FUNCTION_BLOCK FB_RecipeBuilderWings EXTENDS FB_PackML_BaseModule IMPLEMENTS I_RecipeBuilder

VAR
    RecipeBuilder_HMI		: ST_RecipeBuilder_HMI;
    _Config                 : ST_RecipeBuilder_Config;
    _PanelFrontLength       : REAL;  
    _PanelFrontWidth        : REAL;      
    _PanelHeight            : REAL;    
    _RailHeightCorrection   : REAL;

    // --- NOWE ZMIENNE DO PRZECHOWYWANIA SEGMENTÓW ---
    _SegmentsCutX           : ARRAY [1..32] OF ST_CutSegment;
    _SegmentsCutY           : ARRAY [1..32] OF ST_CutSegment;
    _SegmentsGroove         : ARRAY [1..32] OF ST_CutSegment;
    _SegmentsToCutX         : INT;
    _SegmentsToCutY         : INT;
    _SegmentsToGroove       : INT;
END_VAR

METHOD Build : BOOL
VAR
    TotalY          : REAL;
    TotalX          : REAL;
    ShorterY        : REAL;
    ShorterX        : REAL;
    
    // Zmienna lokalna, dopóki nie dodasz jej do ST_RecipeBuilder_Config
    CuttingOverpass : REAL := 20.0; 
END_VAR

// Wyliczenia gabarytów na podstawie parametrów wejściowych (ze struktury _Config)
TotalY   := _Config.PanelFrontLength + 2 * _Config.PanelHeight;
TotalX   := _Config.PanelFrontWidht  + 2 * _Config.PanelHeight; // Uwaga na literówkę 'Widht' w strukturze!
ShorterY := TotalY - _Config.PanelHeight;
ShorterX := TotalX - _Config.PanelHeight;

// --- TRACE DLA WERYFIKACJI ---
Trace(Message:= CONCAT('--- BUILD BORGO WINGS START ---', ''));
Trace(Message:= CONCAT('Input PanelWidth: ', TO_STRING(_Config.PanelFrontWidht)));
Trace(Message:= CONCAT('Input PanelLength: ', TO_STRING(_Config.PanelFrontLength)));
Trace(Message:= CONCAT('Input PanelHeight: ', TO_STRING(_Config.PanelHeight)));
Trace(Message:= CONCAT('Calc TotalX: ', TO_STRING(TotalX)));
Trace(Message:= CONCAT('Calc TotalY: ', TO_STRING(TotalY)));
Trace(Message:= CONCAT('Calc ShorterX: ', TO_STRING(ShorterX)));
Trace(Message:= CONCAT('Calc ShorterY: ', TO_STRING(ShorterY)));

// ------------------------------------
// 1. Segregracja frezowania (Grooving)
// ------------------------------------
_SegmentsToGroove := 4;

_SegmentsGroove[1].Start.X := TotalX;
_SegmentsGroove[1].Stop.X  := 0;
_SegmentsGroove[1].Start.Y := ShorterY;
_SegmentsGroove[1].Stop.Y  := ShorterY;

_SegmentsGroove[2].Start.X := TotalX;
_SegmentsGroove[2].Stop.X  := 0; 
_SegmentsGroove[2].Start.Y := _Config.PanelHeight;
_SegmentsGroove[2].Stop.Y  := _Config.PanelHeight;

_SegmentsGroove[3].Start.X := ShorterX;
_SegmentsGroove[3].Stop.X  := ShorterX;
_SegmentsGroove[3].Start.Y := TotalY;
_SegmentsGroove[3].Stop.Y  := 0;

_SegmentsGroove[4].Start.Y := TotalY;
_SegmentsGroove[4].Stop.Y  := 0;
_SegmentsGroove[4].Start.X := _Config.PanelHeight;
_SegmentsGroove[4].Stop.X  := _Config.PanelHeight;

// ------------------------------------
// 2. Cięcie w osi X (Cut X)
// ------------------------------------
_SegmentsToCutX := 6;

// Short Box Segments
_SegmentsCutX[1].Start.X := TotalX + CuttingOverpass;
_SegmentsCutX[1].Stop.X  := ShorterX;
_SegmentsCutX[1].Start.Y := ShorterY;
_SegmentsCutX[1].Stop.Y  := ShorterY;

_SegmentsCutX[2].Start.X := _Config.PanelHeight;
_SegmentsCutX[2].Stop.X  := -CuttingOverpass;
_SegmentsCutX[2].Start.Y := ShorterY;
_SegmentsCutX[2].Stop.Y  := ShorterY;

_SegmentsCutX[3].Start.X := TotalX + CuttingOverpass;
_SegmentsCutX[3].Stop.X  := ShorterX;
_SegmentsCutX[3].Start.Y := _Config.PanelHeight;
_SegmentsCutX[3].Stop.Y  := _Config.PanelHeight;

_SegmentsCutX[4].Start.X := _Config.PanelHeight;
_SegmentsCutX[4].Stop.X  := -CuttingOverpass;
_SegmentsCutX[4].Start.Y := _Config.PanelHeight;
_SegmentsCutX[4].Stop.Y  := _Config.PanelHeight;

// Panel Dimensions Shorter Flaps
_SegmentsCutX[5].Start.X := TotalX + CuttingOverpass;
_SegmentsCutX[5].Stop.X  := -CuttingOverpass;
_SegmentsCutX[5].Start.Y := TotalY - _Config.RailHeightCorrection;
_SegmentsCutX[5].Stop.Y  := TotalY - _Config.RailHeightCorrection;

_SegmentsCutX[6].Start.X := TotalX + CuttingOverpass;
_SegmentsCutX[6].Stop.X  := -CuttingOverpass;
_SegmentsCutX[6].Start.Y := _Config.RailHeightCorrection;
_SegmentsCutX[6].Stop.Y  := _Config.RailHeightCorrection;

// ------------------------------------
// 3. Cięcie w osi Y (Cut Y)
// ------------------------------------
_SegmentsToCutY := 6;

// Short Box Segments
_SegmentsCutY[1].Start.X := ShorterX;
_SegmentsCutY[1].Stop.X  := ShorterX;
_SegmentsCutY[1].Start.Y := TotalY + CuttingOverpass;
_SegmentsCutY[1].Stop.Y  := ShorterY;

_SegmentsCutY[2].Start.X := _Config.PanelHeight;
_SegmentsCutY[2].Stop.X  := _Config.PanelHeight;
_SegmentsCutY[2].Start.Y := TotalY + CuttingOverpass;
_SegmentsCutY[2].Stop.Y  := ShorterY;

_SegmentsCutY[3].Start.X := ShorterX;
_SegmentsCutY[3].Stop.X  := ShorterX;
_SegmentsCutY[3].Start.Y := _Config.PanelHeight;
_SegmentsCutY[3].Stop.Y  := -CuttingOverpass;

_SegmentsCutY[4].Start.X := _Config.PanelHeight;
_SegmentsCutY[4].Stop.X  := _Config.PanelHeight;
_SegmentsCutY[4].Start.Y := _Config.PanelHeight;
_SegmentsCutY[4].Stop.Y  := -CuttingOverpass;

// Panel Dimensions
_SegmentsCutY[5].Start.X := TotalX;
_SegmentsCutY[5].Stop.X  := TotalX;
_SegmentsCutY[5].Start.Y := TotalY + CuttingOverpass;
_SegmentsCutY[5].Stop.Y  := -CuttingOverpass;

_SegmentsCutY[6].Start.X := 0;
_SegmentsCutY[6].Stop.X  := 0;
_SegmentsCutY[6].Start.Y := TotalY + CuttingOverpass;
_SegmentsCutY[6].Stop.Y  := -CuttingOverpass;

// Log podsumowujący ile odcinków wygenerowano
Trace(Message:= CONCAT('Segments Groove Count: ', TO_STRING(_SegmentsToGroove)));
Trace(Message:= CONCAT('Segments CutX Count: ', TO_STRING(_SegmentsToCutX)));
Trace(Message:= CONCAT('Segments CutY Count: ', TO_STRING(_SegmentsToCutY)));

//Zwracamy TRUE gdy budowanie się zakończyło
Build := TRUE;
END_METHOD

PROPERTY Config : ST_RecipeBuilder_Config
GET
Config := _Config;
END_GET
SET
RecipeBuilder_HMI.Config := Config;
END_SET
END_PROPERTY

// Provides interlocks for HMI control and updates HMI status information for this module
METHOD PROTECTED HMICommunication

// This method is called cyclically by CyclicLogic()
_PanelFrontWidth      := RecipeBuilder_HMI.Config.PanelFrontWidht;
_PanelFrontLength     := RecipeBuilder_HMI.Config.PanelFrontLength;
_PanelHeight          := RecipeBuilder_HMI.Config.PanelHeight;
_RailHeightCorrection := RecipeBuilder_HMI.Config.RailHeightCorrection;
END_METHOD

PROPERTY SegmentsCutX : REFERENCE TO ARRAY [1..32] OF ST_CutSegment
GET
SegmentsCutX REF= _SegmentsCutX;
END_GET
END_PROPERTY

PROPERTY SegmentsCutY : REFERENCE TO ARRAY [1..32] OF ST_CutSegment
GET
SegmentsCutY REF= _SegmentsCutY;
END_GET
END_PROPERTY

PROPERTY SegmentsGroove : REFERENCE TO ARRAY [1..32] OF ST_CutSegment
GET
SegmentsGroove REF= _SegmentsGroove;
END_GET
END_PROPERTY


PROPERTY SegmentsToCutX : INT
GET
SegmentsToCutX := _SegmentsToCutX;
END_GET
END_PROPERTY


PROPERTY SegmentsToCutY : INT
GET
SegmentsToCutY := _SegmentsToCutY;
END_GET
END_PROPERTY


PROPERTY SegmentsToGroove : INT
GET
SegmentsToGroove := _SegmentsToGroove;
END_GET
END_PROPERTY

END_FUNCTION_BLOCK

(* stored: Version 1.1.0.1, ProductVersion 3.1.4024.15
   POU FB_RecipeBuilderWings: Id {3f83a514-1f2f-4e3d-921c-ca7c0b60e17f}, SpecialFunc None
   Method Build: Id {c08ade7c-db75-4c50-8457-5bb392619adf}
   Property Config: Id {e53be9fd-6b88-49c9-8736-ae6ec54e43d8}
   Get Get: Id {0bd9a01b-52a6-47dd-b6fc-d6ccf0a489a9}
   Set Set: Id {e2eb298e-f304-4e9d-ab04-77a183356e49}
   Method HMICommunication: Id {5b58a0e6-30db-439b-a833-a33f4b223005}
   Property SegmentsCutX: Id {9152e646-9866-44c9-b9e6-5a764990d7d4}
   Get Get: Id {8272f94b-fbfa-4156-a332-efb73ed5cf2e}
   Property SegmentsCutY: Id {255ca92b-c547-401c-9784-b32df54e5e2a}
   Get Get: Id {4b559848-f1de-4c18-834d-4d2909a2699d}
   Property SegmentsGroove: Id {a6cc8c84-07e4-4531-824b-69c46a3f14a3}
   Get Get: Id {7a846cca-77b5-4d85-b851-6d33d3df4235}
   Property SegmentsToCutX: Id {e45efa5d-ccfc-458e-9811-5f080acfb1d1}
   Get Get: Id {58e9fc3c-a2ea-47ff-862f-fb085769cffc}
   Property SegmentsToCutY: Id {0f05ab0b-f50d-4ba7-9a3d-ced7155bbd03}
   Get Get: Id {dd01e30b-5156-462c-981f-e1777bde948b}
   Property SegmentsToGroove: Id {e4a3954d-3a1b-4d86-a891-2e859afd79f8}
   Get Get: Id {166af98c-be7e-4a9c-8000-ac82596ec13a} *)
